FUNCTION_BLOCK Motor
VAR_INPUT
	velocity : INT;
END_VAR
VAR_OUTPUT
	counter : UINT;
END_VAR
VAR PERSISTENT
	internalCounter : UINT;
END_VAR

internalCounter := internalCounter + velocity*10;
counter := internalCounter;

END_FUNCTION_BLOCK

(* stored: Version 1.1.0.1, ProductVersion 3.1.4024.10
   POU Motor: Id {710e4976-0d7b-4351-b5ec-7ccf087d8b32}, SpecialFunc None *)
